PROGRAM OnGantry_IO
VAR
	//watchdog
	intBoneCounter	:INT	:=0;
	tonSwReset :TON;
	tpSwReset :Tp;
	
	//Interface of IO To RTC		
	plc_to_io_bGantryTouchGuard   AT%I*   : BOOL;
	plc_to_cpp_bGantryTouchGuard  AT%Q*   : BOOL;
	
	plc_to_io_bAutoMove           AT%I*   : BOOL;
	plc_to_cpp_bAutoMove          AT%Q*   : BOOL;
	
	plc_to_io_OnGantryRtcWdOK     AT%I*   : BOOL;
	plc_to_cpp_OnGantryRtcWdOK    AT%Q*   : BOOL;
	
	plc_to_io_bCanOpenOk          AT%Q*   : BOOL;
	plc_to_cpp_bCanOpenOk         AT%I*   : BOOL;
		
	plc_to_io_OnGantryMoveEn      AT%Q*   : BOOL;
	plc_to_cpp_OnGantryMoveEn     AT%I*   : BOOL;
		
	plc_to_io_bSwWatchDogService  AT%Q*   : BOOL;
	
	plc_to_io_bSwRest             AT%Q*   : BOOL;
	plc_to_cpp_bSwRest            AT%I*   : BOOL;
	
	plc_to_io_bKvEn               AT%Q*   : BOOL;
	plc_to_cpp_bKvEn              AT%I*   : BOOL;
	
	plc_to_io_bEthercatInOk       AT%Q*   : BOOL;
	plc_to_cpp_bEthercatInOk      AT%I*   : BOOL;
	
	plc_to_io_bEthercatOutOk      AT%Q*   : BOOL;
	plc_to_cpp_bEthercatOutOk     AT%I*   : BOOL;	
	
	plc_to_cpp_bSwManualMotionEn  AT%I*		:BOOL;
	plc_to_io_bSwManualMotionEn   AT%Q*		:BOOL;
END_VAR

IF intBoneCounter >= 4 THEN
	plc_to_io_bSwWatchDogService := NOT plc_to_io_bSwWatchDogService;		//Flip bone to feed the dog
	intBoneCounter := 0;
ELSE intBoneCounter := intBoneCounter + 1; 
END_IF

IF plc_to_io_bSwRest AND (NOT plc_to_cpp_bSwRest) THEN		// turn io signal to false in next cycle if cpp signal is false
	plc_to_io_bSwRest := FALSE;
END_IF

tpSwReset(IN:=TwinCAT_SystemInfoVarList._TaskInfo[Tc2_System.GETCURTASKINDEXEX()].FirstCycle,PT:=T#2S,Q=>,ET=>);
tonSwReset(IN:=tpSwReset.Q,PT:=T#1S,Q=>,ET=>);		//Reset pulse will send after 1sec of PLC first cycle

plc_to_io_bSwRest := plc_to_cpp_bSwRest OR tonSwReset.Q;

io_update();

ACTION io_update:


////****beta interface of plc and cpp****////
//inputIO to plc to cpp	
plc_to_cpp_bGantryTouchGuard := plc_to_io_bGantryTouchGuard;
plc_to_cpp_bAutoMove := plc_to_io_bAutoMove;        
plc_to_cpp_OnGantryRtcWdOK  := plc_to_io_OnGantryRtcWdOK ;
     
     
plc_to_io_bCanOpenOk :=	plc_to_cpp_bCanOpenOk;
plc_to_io_OnGantryMoveEn := plc_to_cpp_OnGantryMoveEn;    	
plc_to_io_bSwRest := plc_to_cpp_bSwRest;          	         	
plc_to_io_bKvEn :=  plc_to_cpp_bKvEn;        
plc_to_io_bEthercatOutOk := plc_to_cpp_bEthercatOutOk;
plc_to_io_bEthercatInOk := plc_to_cpp_bEthercatInOk; 

plc_to_io_bSwManualMotionEn:=plc_to_cpp_bSwManualMotionEn;
END_ACTION

END_PROGRAM

(* stored: Version 1.1.0.1, ProductVersion 3.1.4022.10
   POU OnGantry_IO: Id {5422ddab-74cb-416c-81ac-d1795660be07}, SpecialFunc None
   Action io_update: Id {9dadd95c-93d6-4d40-a7ba-5efc22ba5c10} *)
